// TIA Portal V21 export
TYPE "LBC_Basic_typeAnalogOutputConfiguration"
TITLE = LBC_typeAnalogOutputConfiguration_Basic
// Module related configuration parameters
   STRUCT
      referenceDesignator { S7_SetPoint := 'True'} : WString := WSTRING#'AnalogOutput';   // Device name or device ID
      physicalUnit { S7_SetPoint := 'True'} : String[10] := 'unit';   // Each value should have a physical unit (like [°C], [kWh], etc.)
      isUnipolarSignal { S7_SetPoint := 'True'} : Bool := TRUE;   // TRUE: Sensor is a unipolar type (just positive values), FALSE: Sensor is a bipolar type (positive and negative values)
      default { S7_SetPoint := 'True'} : Int := 0;   // Default OUTPUT analog value to be returned if function block is not enabled or quality is bad
      limitHigh { S7_SetPoint := 'True'} : LReal := 80.0;   // Process value limit high 1
      limitLow { S7_SetPoint := 'True'} : LReal := -80.0;   // Process value limit low 1
      processValueMax { S7_SetPoint := 'True'} : LReal := 100.0;   // Maximum limit of the process value
      processValueMin { S7_SetPoint := 'True'} : LReal := -100.0;   // Minimum limit of the process value
      scaleProcessUppPoint { S7_SetPoint := 'True'} : LReal := 100.0;   // Upper point for the process value
      scaleProcessLowPoint { S7_SetPoint := 'True'} : LReal := -100.0;   // Lower point for the process value
      scaleAnalogUppPoint { S7_SetPoint := 'True'} : LReal := 27648.0;   // Upper point for the analog output. Maximum value from the hardware module - i.e. 27648 - scaled value
      scaleAnalogLowPoint { S7_SetPoint := 'True'} : LReal := 0.0;   // Lower point for the analog output. Minimum value from the hardware module - i.e. 0 - scaled value
   END_STRUCT;
END_TYPE
